// TIA Portal project "CLP_Simulator" (V17)

(* hardware
DEVICE "S7-1500/ET200MP station_1"  S7-1500 station
   slot 0: "Rail_0"  Rack  6ES7 590-1***0-0AA0
   slot 1: "S71500_Sim"  CPU 1513-1 PN  6ES7 513-1AL02-0AB0  V2.9
      slot 3: "CPU display_1"  6ES7591-1AA00-0AA0
      slot 32768: "PROFINET interface_1"  X1
         slot 32769: "Port_1"  X1 P1
         slot 32770: "Port_2"  X1 P2
      slot 34817: "Virtual CP interface port_1"  Virtual CP interface port  Virtual CP interface port
DEVICE "S7-1200 station_1"  S7-1200 Station
   slot 0: "Rack_0"  S7-1200 Rack  Rack  V1.0
   slot 1: "S71200_Real"  CPU 1214C DC/DC/DC  6ES7 214-1AE30-0XB0  V2.2
*)

// ===== PLC "S71500_Sim"  CPU 1513-1 PN =====

VAR_GLOBAL   // PLC tag table "Default tag table"
   "System_Byte" AT %MB1000 : Byte;
   "FirstScan" AT %M1000.0 : Bool;
   "DiagStatusUpdate" AT %M1000.1 : Bool;
   "AlwaysTRUE" AT %M1000.2 : Bool;
   "AlwaysFALSE" AT %M1000.3 : Bool;
   "Clock_Byte" AT %MB1001 : Byte;
   "Clock_10Hz" AT %M1001.0 : Bool;
   "Clock_5Hz" AT %M1001.1 : Bool;
   "Clock_2.5Hz" AT %M1001.2 : Bool;
   "Clock_2Hz" AT %M1001.3 : Bool;
   "Clock_1.25Hz" AT %M1001.4 : Bool;
   "Clock_1Hz" AT %M1001.5 : Bool;
   "Clock_0.625Hz" AT %M1001.6 : Bool;
   "Clock_0.5Hz" AT %M1001.7 : Bool;
   "Valor_1" AT %MW0 : Int;
   "Valor2" AT %MD10 : Real;
   "Valor_3" AT %MD6 : Real;
END_VAR

DATA_BLOCK "Fail_Generators"   // DB10
{ S7_Optimized_Access := 'FALSE' }
VERSION : 0.1
   VAR
      Kill_Bateria : Bool;
      Kill_PV : Bool;
      Kill_AC_Output : Bool;
   END_VAR
BEGIN
END_DATA_BLOCK

DATA_BLOCK "Inversor_Multiplus"   // DB49
{ S7_Optimized_Access := 'FALSE' }
VERSION : 0.1
   VAR
      "." : Real;
      ".." : Real;
      "..." : Real;
      "....." : Real;
      "......" : Real;
      "......." : Real;
      Current_Out : Real := 17.45;
      Voltage_Out : Real := 220.3;
   END_VAR
BEGIN
END_DATA_BLOCK

DATA_BLOCK "Controlador_Carga"   // DB50
{ S7_Optimized_Access := 'FALSE' }
VERSION : 0.1
   VAR
      PV_Power_In : Real := 1.0;
      Current_Bus : Real := 2.0;
      Voltage_Bus : Real := 3.0;
      Max_Power_Today : Real := 4.0;
      "." : Real;
      Yield_Diario : Real := 5.0;
   END_VAR
BEGIN
END_DATA_BLOCK

DATA_BLOCK "BateriaBYD"   // DB51
{ S7_Optimized_Access := 'FALSE' }
VERSION : 0.1
   VAR
      Current : Real := 10.0;
      "." : Real;
      Voltage : Real := 20.0;
      Carga_Bateria : Real := 25.5;
   END_VAR
BEGIN
END_DATA_BLOCK

DATA_BLOCK "Medidor_Analisador"   // DB52
{ S7_Optimized_Access := 'FALSE' }
VERSION : 0.1
   VAR
      Current_R_Med : Real := 1.0;
      Current_S_Med : Real := 1.0;
      Current_T_Med : Real := 1.0;
      Current_N_Med : Real := 1.0;
      "." : Real;
      "._1" : Real;
      "._2" : Real;
      "._3" : Real;
      "._4" : Real;
      "._5" : Real;
      "._6" : Real;
      "._7" : Real;
      "._8" : Real;
      "._9" : Real;
      "._10" : Real;
      "._11" : Real;
      "._12" : Real;
      "._13" : Real;
      "._14" : Real;
      "._15" : Real;
      "._1_1" : Real;
      "._2_1" : Real;
      "._3_1" : Real;
      "._4_1" : Real;
      "._5_1" : Real;
      "._6_1" : Real;
      "._7_1" : Real;
      "._8_1" : Real;
      "._9_1" : Real;
      "._10_1" : Real;
      "._1_2" : Real;
      "._2_2" : Real;
      "._3_2" : Real;
      "._4_2" : Real;
      "._5_2" : Real;
      "._6_2" : Real;
      "._7_2" : Real;
      "._8_2" : Real;
      "._9_2" : Real;
      Current_L1N_Ana : Real := 1.0;
      Current_L2N_Ana : Real := 1.0;
      Current_L3N_Ana : Real := 1.0;
      "._3_3" : Real;
      Power_Sys_Ana : Real := 1.0;
   END_VAR
BEGIN
END_DATA_BLOCK

// folder: System blocks/Program resources

DATA_BLOCK "Sim_Cycle_DB"   // DB1
{ S7_Optimized_Access := 'TRUE' }
AUTHOR : SIMATIC
FAMILY : IEC
NAME : DCNTR
VERSION : 1.2
// stored: InstanceOfName IEC_DCOUNTER
"IEC_DCOUNTER"
BEGIN
END_DATA_BLOCK

// folder: (top level)

ORGANIZATION_BLOCK "Main"   // OB1, LAD, ProgramCycle
TITLE = "Main Program Sweep (Cycle)"
{ S7_Optimized_Access := 'TRUE' }
VERSION : 0.1
   VAR_INPUT
      Initial_Call : Bool;   // Initial call of this OB
      Remanence : Bool;   // =True, if remanent data are available
   END_VAR
   VAR_TEMP
      fast_noise : Int;
      rad_time_of_day : Real;
      pv_power_total : Real;
      rad_cycle : Real;
   END_VAR
BEGIN

REGION Network 1: Generators
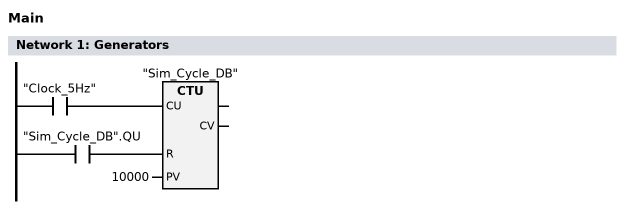
   "Sim_Cycle_DB".CTU(CU := "Clock_5Hz", R := "Sim_Cycle_DB".QU, PV := 10000);
END_REGION

REGION Network 2 (SCL): Simulação e Atribuição
   REGION "Motor de Simulação"
       #rad_cycle := DINT_TO_REAL("Sim_Cycle_DB".CV) * 0.01;
   END_REGION


   REGION "DB51: BateriaBYD"
       IF "Fail_Generators"."Kill_Bateria" THEN
           "BateriaBYD"."Voltage" := 0.0;
           "BateriaBYD"."Current" := 0.0;
       ELSE
           // Tensão (Range: 51.5 a 52.5 V)
           "BateriaBYD"."Voltage" := 52.0 + (0.5 * SIN(#rad_cycle * 0.2));
           // Corrente (Range: -50.0 a +50.0 A)
           "BateriaBYD"."Current" := 0.0 + (50.0 * SIN(#rad_cycle * 0.5));
       END_IF;

       // Carga (SOC) não é tensão/corrente, então continua oscilando
       "BateriaBYD"."Carga_Bateria" := 60.0 + (40.0 * SIN(#rad_cycle * 0.1));
   END_REGION


   REGION "DB50: Controlador_Carga"
       // --- Potência Solar ---
       IF "Fail_Generators"."Kill_PV" THEN
           "Controlador_Carga"."PV_Power_In" := 0.0;
       ELSE
           // Potência Solar (Range: 0.0 a 8000.0 W)
           "Controlador_Carga"."PV_Power_In" := (SIN(#rad_cycle * 0.3) + 1.0) * 4000.0;
       END_IF;

       // --- Tensão do Barramento DC ---
       // O barramento DC é mantido pela Bateria. Se a bateria for morta, o barramento também morre.
       IF "Fail_Generators"."Kill_Bateria" THEN
           "Controlador_Carga"."Voltage_Bus" := 0.0;
       ELSE
           "Controlador_Carga"."Voltage_Bus" := 58.5 + (0.5 * SIN(#rad_cycle * 0.4));
       END_IF;

       // --- Corrente do Barramento DC (I = P / V) ---
       // Esta lógica se auto-corrige: Se PV_Power_In for 0, Current_Bus será 0.
       IF "Controlador_Carga"."Voltage_Bus" > 1.0 THEN
           "Controlador_Carga"."Current_Bus" := "Controlador_Carga"."PV_Power_In" / "Controlador_Carga"."Voltage_Bus";
       ELSE
           "Controlador_Carga"."Current_Bus" := 0.0;
       END_IF;

       // Valores de status (não são Tensão/Corrente)
       "Controlador_Carga"."Max_Power_Today" := 7975.0 + (25.0 * SIN(#rad_cycle * 0.05));
       "Controlador_Carga"."Yield_Diario" := DINT_TO_REAL("Sim_Cycle_DB".CV) * 0.005;
   END_REGION


   REGION "DB49: Inversor_Multiplus"
       // --- Saída AC Principal ---
       IF "Fail_Generators"."Kill_AC_Output" THEN
           "Inversor_Multiplus"."Voltage_Out" := 0.0;
           "Inversor_Multiplus"."Current_Out" := 0.0;
       ELSE
           // Tensão de Saída AC (Range: 219.0 a 221.0 V)
           "Inversor_Multiplus"."Voltage_Out" := 220.0 + (1.0 * SIN(#rad_cycle * 0.6));
           // Corrente de Saída AC (Range: 5.0 a 30.0 A)
           "Inversor_Multiplus"."Current_Out" := 17.5 + (12.5 * SIN(#rad_cycle * 0.8));
       END_IF;
   END_REGION


   REGION "DB52: Medidor_Analisador"
       // Se a saída AC do Inversor (fonte) for morta, todas as cargas (correntes) AC morrem.
       IF "Fail_Generators"."Kill_AC_Output" THEN
           "Medidor_Analisador".Current_L1N_Ana := 0.0;
           "Medidor_Analisador".Current_L2N_Ana := 0.0;
           "Medidor_Analisador".Current_L3N_Ana := 0.0;
           "Medidor_Analisador".Current_R_Med := 0.0;
           "Medidor_Analisador".Current_S_Med := 0.0;
           "Medidor_Analisador".Current_T_Med := 0.0;
           "Medidor_Analisador".Current_N_Med := 0.0;
           "Medidor_Analisador".Power_Sys_Ana := 0.0;
       ELSE
           // Correntes das Fases
           "Medidor_Analisador".Current_L1N_Ana := 8.0 + (4.0 * SIN(#rad_cycle * 1.1));
           "Medidor_Analisador".Current_L2N_Ana := 7.0 + (3.0 * SIN(#rad_cycle * 0.9));
           "Medidor_Analisador".Current_L3N_Ana := 9.0 + (5.0 * SIN(#rad_cycle * 1.3));

           "Medidor_Analisador".Current_R_Med := 9.5 + (1.0 * SIN(#rad_cycle * 1.5));
           "Medidor_Analisador".Current_S_Med := 10.3 + (1.0 * SIN(#rad_cycle * 1.5));
           "Medidor_Analisador".Current_T_Med := 11.7 + (1.0 * SIN(#rad_cycle * 1.5));
           "Medidor_Analisador".Current_N_Med := 1.5 + (1.0 * SIN(#rad_cycle * 1.5));

           // Potência Total do Sistema
           "Medidor_Analisador".Power_Sys_Ana := ("Medidor_Analisador".Current_L1N_Ana
           + "Medidor_Analisador".Current_L2N_Ana
           + "Medidor_Analisador".Current_L3N_Ana) * 220.0;
       END_IF;
   END_REGION
END_REGION
END_ORGANIZATION_BLOCK

// ===== PLC "S71200_Real"  CPU 1214C DC/DC/DC =====

VAR_GLOBAL   // PLC tag table "Default tag table"
   "System_Byte" AT %MB1000 : Byte;
   "FirstScan" AT %M1000.0 : Bool;
   "DiagStatusUpdate" AT %M1000.1 : Bool;
   "AlwaysTRUE" AT %M1000.2 : Bool;
   "AlwaysFALSE" AT %M1000.3 : Bool;
   "Clock_Byte" AT %MB1001 : Byte;
   "Clock_10Hz" AT %M1001.0 : Bool;
   "Clock_5Hz" AT %M1001.1 : Bool;
   "Clock_2.5Hz" AT %M1001.2 : Bool;
   "Clock_2Hz" AT %M1001.3 : Bool;
   "Clock_1.25Hz" AT %M1001.4 : Bool;
   "Clock_1Hz" AT %M1001.5 : Bool;
   "Clock_0.625Hz" AT %M1001.6 : Bool;
   "Clock_0.5Hz" AT %M1001.7 : Bool;
END_VAR

DATA_BLOCK "Fail_Generators"   // DB10
{ S7_Optimized_Access := 'FALSE' }
VERSION : 0.1
   VAR
      Kill_Bateria : Bool;
      Kill_PV : Bool;
      Kill_AC_Output : Bool;
   END_VAR
BEGIN
END_DATA_BLOCK

DATA_BLOCK "Inversor_Multiplus"   // DB49
{ S7_Optimized_Access := 'FALSE' }
VERSION : 0.1
   VAR
      "." : Real;
      ".." : Real;
      "..." : Real;
      "....." : Real;
      "......" : Real;
      "......." : Real;
      Current_Out : Real := 17.45;
      Voltage_Out : Real := 220.3;
   END_VAR
BEGIN
END_DATA_BLOCK

DATA_BLOCK "Controlador_Carga"   // DB50
{ S7_Optimized_Access := 'FALSE' }
VERSION : 0.1
   VAR
      PV_Power_In : Real := 1.0;
      Current_Bus : Real := 2.0;
      Voltage_Bus : Real := 3.0;
      Max_Power_Today : Real := 4.0;
      "." : Real;
      Yield_Diario : Real := 5.0;
   END_VAR
BEGIN
END_DATA_BLOCK

DATA_BLOCK "BateriaBYD"   // DB51
{ S7_Optimized_Access := 'FALSE' }
VERSION : 0.1
   VAR
      Current : Real := 10.0;
      "." : Real;
      Voltage : Real := 20.0;
      Carga_Bateria : Real := 25.5;
   END_VAR
BEGIN
END_DATA_BLOCK

DATA_BLOCK "Medidor_Analisador"   // DB52
{ S7_Optimized_Access := 'FALSE' }
VERSION : 0.1
   VAR
      Current_R_Med : Real := 1.0;
      Current_S_Med : Real := 1.0;
      Current_T_Med : Real := 1.0;
      Current_N_Med : Real := 1.0;
      "." : Real;
      "._1" : Real;
      "._2" : Real;
      "._3" : Real;
      "._4" : Real;
      "._5" : Real;
      "._6" : Real;
      "._7" : Real;
      "._8" : Real;
      "._9" : Real;
      "._10" : Real;
      "._11" : Real;
      "._12" : Real;
      "._13" : Real;
      "._14" : Real;
      "._15" : Real;
      "._1_1" : Real;
      "._2_1" : Real;
      "._3_1" : Real;
      "._4_1" : Real;
      "._5_1" : Real;
      "._6_1" : Real;
      "._7_1" : Real;
      "._8_1" : Real;
      "._9_1" : Real;
      "._10_1" : Real;
      "._1_2" : Real;
      "._2_2" : Real;
      "._3_2" : Real;
      "._4_2" : Real;
      "._5_2" : Real;
      "._6_2" : Real;
      "._7_2" : Real;
      "._8_2" : Real;
      "._9_2" : Real;
      Current_L1N_Ana : Real := 1.0;
      Current_L2N_Ana : Real := 1.0;
      Current_L3N_Ana : Real := 1.0;
      "._3_3" : Real;
      Power_Sys_Ana : Real := 1.0;
   END_VAR
BEGIN
END_DATA_BLOCK

// folder: System blocks/Program resources

DATA_BLOCK "Sim_Cycle_DB"   // DB1
{ S7_Optimized_Access := 'TRUE' }
AUTHOR : Simatic
FAMILY : IEC
NAME : CNTR
VERSION : 1.0
// stored: InstanceOfName IEC_COUNTER
"IEC_COUNTER"
BEGIN
END_DATA_BLOCK

// folder: (top level)

ORGANIZATION_BLOCK "Main"   // OB1, LAD, ProgramCycle
TITLE = "Main Program Sweep (Cycle)"
{ S7_Optimized_Access := 'TRUE' }
VERSION : 0.1
   VAR_TEMP
      fast_noise : Int;
      rad_time_of_day : Real;
      pv_power_total : Real;
      rad_cycle : Real;
   END_VAR
BEGIN

REGION Network 1: Generators
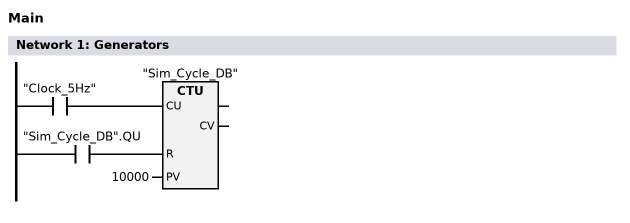
   "Sim_Cycle_DB".CTU(CU := "Clock_5Hz", R := "Sim_Cycle_DB".QU, PV := 10000);
END_REGION

REGION Network 2 (SCL): Simulação e Atribuição
   REGION "Motor de Simulação"
       #rad_cycle := DINT_TO_REAL("Sim_Cycle_DB".CV) * 0.01;
   END_REGION


   REGION "DB51: BateriaBYD"
       IF "Fail_Generators"."Kill_Bateria" THEN
           "BateriaBYD"."Voltage" := 0.0;
           "BateriaBYD"."Current" := 0.0;
       ELSE
           // Tensão (Range: 51.5 a 52.5 V)
           "BateriaBYD"."Voltage" := 52.0 + (0.5 * SIN(#rad_cycle * 0.2));
           // Corrente (Range: -50.0 a +50.0 A)
           "BateriaBYD"."Current" := 0.0 + (50.0 * SIN(#rad_cycle * 0.5));
       END_IF;

       // Carga (SOC) não é tensão/corrente, então continua oscilando
       "BateriaBYD"."Carga_Bateria" := 60.0 + (40.0 * SIN(#rad_cycle * 0.1));
   END_REGION


   REGION "DB50: Controlador_Carga"
       // --- Potência Solar ---
       IF "Fail_Generators"."Kill_PV" THEN
           "Controlador_Carga"."PV_Power_In" := 0.0;
       ELSE
           // Potência Solar (Range: 0.0 a 8000.0 W)
           "Controlador_Carga"."PV_Power_In" := (SIN(#rad_cycle * 0.3) + 1.0) * 4000.0;
       END_IF;

       // --- Tensão do Barramento DC ---
       // O barramento DC é mantido pela Bateria. Se a bateria for morta, o barramento também morre.
       IF "Fail_Generators"."Kill_Bateria" THEN
           "Controlador_Carga"."Voltage_Bus" := 0.0;
       ELSE
           "Controlador_Carga"."Voltage_Bus" := 58.5 + (0.5 * SIN(#rad_cycle * 0.4));
       END_IF;

       // --- Corrente do Barramento DC (I = P / V) ---
       // Esta lógica se auto-corrige: Se PV_Power_In for 0, Current_Bus será 0.
       IF "Controlador_Carga"."Voltage_Bus" > 1.0 THEN
           "Controlador_Carga"."Current_Bus" := "Controlador_Carga"."PV_Power_In" / "Controlador_Carga"."Voltage_Bus";
       ELSE
           "Controlador_Carga"."Current_Bus" := 0.0;
       END_IF;

       // Valores de status (não são Tensão/Corrente)
       "Controlador_Carga"."Max_Power_Today" := 7975.0 + (25.0 * SIN(#rad_cycle * 0.05));
       "Controlador_Carga"."Yield_Diario" := DINT_TO_REAL("Sim_Cycle_DB".CV) * 0.005;
   END_REGION


   REGION "DB49: Inversor_Multiplus"
       // --- Saída AC Principal ---
       IF "Fail_Generators"."Kill_AC_Output" THEN
           "Inversor_Multiplus"."Voltage_Out" := 0.0;
           "Inversor_Multiplus"."Current_Out" := 0.0;
       ELSE
           // Tensão de Saída AC (Range: 219.0 a 221.0 V)
           "Inversor_Multiplus"."Voltage_Out" := 220.0 + (1.0 * SIN(#rad_cycle * 0.6));
           // Corrente de Saída AC (Range: 5.0 a 30.0 A)
           "Inversor_Multiplus"."Current_Out" := 17.5 + (12.5 * SIN(#rad_cycle * 0.8));
       END_IF;
   END_REGION


   REGION "DB52: Medidor_Analisador"
       // Se a saída AC do Inversor (fonte) for morta, todas as cargas (correntes) AC morrem.
       IF "Fail_Generators"."Kill_AC_Output" THEN
           "Medidor_Analisador".Current_L1N_Ana := 0.0;
           "Medidor_Analisador".Current_L2N_Ana := 0.0;
           "Medidor_Analisador".Current_L3N_Ana := 0.0;
           "Medidor_Analisador".Current_R_Med := 0.0;
           "Medidor_Analisador".Current_S_Med := 0.0;
           "Medidor_Analisador".Current_T_Med := 0.0;
           "Medidor_Analisador".Current_N_Med := 0.0;
           "Medidor_Analisador".Power_Sys_Ana := 0.0;
       ELSE
           // Correntes das Fases
           "Medidor_Analisador".Current_L1N_Ana := 8.0 + (4.0 * SIN(#rad_cycle * 1.1));
           "Medidor_Analisador".Current_L2N_Ana := 7.0 + (3.0 * SIN(#rad_cycle * 0.9));
           "Medidor_Analisador".Current_L3N_Ana := 9.0 + (5.0 * SIN(#rad_cycle * 1.3));

           "Medidor_Analisador".Current_R_Med := 9.5 + (1.0 * SIN(#rad_cycle * 1.5));
           "Medidor_Analisador".Current_S_Med := 10.3 + (1.0 * SIN(#rad_cycle * 1.5));
           "Medidor_Analisador".Current_T_Med := 11.7 + (1.0 * SIN(#rad_cycle * 1.5));
           "Medidor_Analisador".Current_N_Med := 1.5 + (1.0 * SIN(#rad_cycle * 1.5));

           // Potência Total do Sistema
           "Medidor_Analisador".Power_Sys_Ana := ("Medidor_Analisador".Current_L1N_Ana
           + "Medidor_Analisador".Current_L2N_Ana
           + "Medidor_Analisador".Current_L3N_Ana) * 220.0;
       END_IF;
   END_REGION
END_REGION
END_ORGANIZATION_BLOCK